FUNCTION_BLOCK FB_HMI_HEATERS EXTENDS FB_HMI_COMPONENT
VAR_INPUT
END_VAR
VAR_OUTPUT
END_VAR
VAR
END_VAR

END_FUNCTION_BLOCK

(* stored: Version 1.1.0.1, ProductVersion 3.1.4024.14
   POU FB_HMI_HEATERS: Id {367b2c7c-470b-486f-a7f5-ebd87b06ceb2}, SpecialFunc None *)
